{attribute 'qualified_only'}
VAR_GLOBAL INTERNAL
	iFirstInit			: I_InitNode;
	iLastInit			: I_InitNode;

	iFirstCyclic		: I_ExecuteNode;
	iLastCyclic			: I_ExecuteNode;
	
	bInit				: BOOL := TRUE;
END_VAR

(* stored: Version 1.1.0.1
   GVL _Runtime: Id {a8108114-c7a2-455b-babd-f14b1e02d6df} *)
